FUNCTION BITS_TO_LWORD
  (* Standard: 61499-1 *)
  (* Version 1.0, 2024-02-22, franz *)
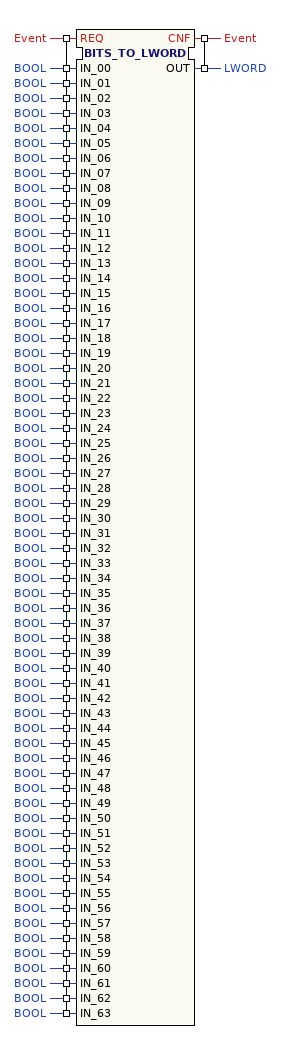
  EVENT_INPUT
    REQ WITH IN_00, IN_01, IN_02, IN_03, IN_04, IN_05, IN_06, IN_07, IN_08, IN_09, IN_10, IN_11, IN_12, IN_13, IN_14, IN_15, IN_16, IN_17, IN_18, IN_19, IN_20, IN_21, IN_22, IN_23, IN_24, IN_25, IN_26, IN_27, IN_28, IN_29, IN_30, IN_31, IN_32, IN_33, IN_34, IN_35, IN_36, IN_37, IN_38, IN_39, IN_40, IN_41, IN_42, IN_43, IN_44, IN_45, IN_46, IN_47, IN_48, IN_49, IN_50, IN_51, IN_52, IN_53, IN_54, IN_55, IN_56, IN_57, IN_58, IN_59, IN_60, IN_61, IN_62, IN_63;
  END_EVENT
  EVENT_OUTPUT
    CNF WITH OUT;
  END_EVENT
  VAR_INPUT
    IN_00 : BOOL; (* BIT 00 *)
    IN_01 : BOOL; (* BIT 01 *)
    IN_02 : BOOL; (* BIT 02 *)
    IN_03 : BOOL; (* BIT 03 *)
    IN_04 : BOOL; (* BIT 04 *)
    IN_05 : BOOL; (* BIT 05 *)
    IN_06 : BOOL; (* BIT 06 *)
    IN_07 : BOOL; (* BIT 07 *)
    IN_08 : BOOL; (* BIT 08 *)
    IN_09 : BOOL; (* BIT 09 *)
    IN_10 : BOOL; (* BIT 10 *)
    IN_11 : BOOL; (* BIT 11 *)
    IN_12 : BOOL; (* BIT 12 *)
    IN_13 : BOOL; (* BIT 13 *)
    IN_14 : BOOL; (* BIT 14 *)
    IN_15 : BOOL; (* BIT 15 *)
    IN_16 : BOOL; (* BIT 16 *)
    IN_17 : BOOL; (* BIT 17 *)
    IN_18 : BOOL; (* BIT 18 *)
    IN_19 : BOOL; (* BIT 19 *)
    IN_20 : BOOL; (* BIT 20 *)
    IN_21 : BOOL; (* BIT 21 *)
    IN_22 : BOOL; (* BIT 22 *)
    IN_23 : BOOL; (* BIT 23 *)
    IN_24 : BOOL; (* BIT 24 *)
    IN_25 : BOOL; (* BIT 25 *)
    IN_26 : BOOL; (* BIT 26 *)
    IN_27 : BOOL; (* BIT 27 *)
    IN_28 : BOOL; (* BIT 28 *)
    IN_29 : BOOL; (* BIT 29 *)
    IN_30 : BOOL; (* BIT 30 *)
    IN_31 : BOOL; (* BIT 31 *)
    IN_32 : BOOL; (* BIT 32 *)
    IN_33 : BOOL; (* BIT 33 *)
    IN_34 : BOOL; (* BIT 34 *)
    IN_35 : BOOL; (* BIT 35 *)
    IN_36 : BOOL; (* BIT 36 *)
    IN_37 : BOOL; (* BIT 37 *)
    IN_38 : BOOL; (* BIT 38 *)
    IN_39 : BOOL; (* BIT 39 *)
    IN_40 : BOOL; (* BIT 40 *)
    IN_41 : BOOL; (* BIT 41 *)
    IN_42 : BOOL; (* BIT 42 *)
    IN_43 : BOOL; (* BIT 43 *)
    IN_44 : BOOL; (* BIT 44 *)
    IN_45 : BOOL; (* BIT 45 *)
    IN_46 : BOOL; (* BIT 46 *)
    IN_47 : BOOL; (* BIT 47 *)
    IN_48 : BOOL; (* BIT 48 *)
    IN_49 : BOOL; (* BIT 49 *)
    IN_50 : BOOL; (* BIT 50 *)
    IN_51 : BOOL; (* BIT 51 *)
    IN_52 : BOOL; (* BIT 52 *)
    IN_53 : BOOL; (* BIT 53 *)
    IN_54 : BOOL; (* BIT 54 *)
    IN_55 : BOOL; (* BIT 55 *)
    IN_56 : BOOL; (* BIT 56 *)
    IN_57 : BOOL; (* BIT 57 *)
    IN_58 : BOOL; (* BIT 58 *)
    IN_59 : BOOL; (* BIT 59 *)
    IN_60 : BOOL; (* BIT 60 *)
    IN_61 : BOOL; (* BIT 61 *)
    IN_62 : BOOL; (* BIT 62 *)
    IN_63 : BOOL; (* BIT 63 *)
  END_VAR
  VAR_OUTPUT
    OUT : LWORD; (* LWORD Output *)
  END_VAR
  BODY IN ST:
FUNCTION BITS_TO_LWORD

VAR_INPUT
	IN_00 : BOOL;    // BIT 00
	IN_01 : BOOL;    // BIT 01
	IN_02 : BOOL;    // BIT 02
	IN_03 : BOOL;    // BIT 03
	IN_04 : BOOL;    // BIT 04
	IN_05 : BOOL;    // BIT 05
	IN_06 : BOOL;    // BIT 06
	IN_07 : BOOL;    // BIT 07
	IN_08 : BOOL;    // BIT 08
	IN_09 : BOOL;    // BIT 09
	IN_10 : BOOL;    // BIT 10
	IN_11 : BOOL;    // BIT 11
	IN_12 : BOOL;    // BIT 12
	IN_13 : BOOL;    // BIT 13
	IN_14 : BOOL;    // BIT 14
	IN_15 : BOOL;    // BIT 15
	IN_16 : BOOL;    // BIT 16
	IN_17 : BOOL;    // BIT 17
	IN_18 : BOOL;    // BIT 18
	IN_19 : BOOL;    // BIT 19
	IN_20 : BOOL;    // BIT 20
	IN_21 : BOOL;    // BIT 21
	IN_22 : BOOL;    // BIT 22
	IN_23 : BOOL;    // BIT 23
	IN_24 : BOOL;    // BIT 24
	IN_25 : BOOL;    // BIT 25
	IN_26 : BOOL;    // BIT 26
	IN_27 : BOOL;    // BIT 27
	IN_28 : BOOL;    // BIT 28
	IN_29 : BOOL;    // BIT 29
	IN_30 : BOOL;    // BIT 30
	IN_31 : BOOL;    // BIT 31
	IN_32 : BOOL;    // BIT 32
	IN_33 : BOOL;    // BIT 33
	IN_34 : BOOL;    // BIT 34
	IN_35 : BOOL;    // BIT 35
	IN_36 : BOOL;    // BIT 36
	IN_37 : BOOL;    // BIT 37
	IN_38 : BOOL;    // BIT 38
	IN_39 : BOOL;    // BIT 39
	IN_40 : BOOL;    // BIT 40
	IN_41 : BOOL;    // BIT 41
	IN_42 : BOOL;    // BIT 42
	IN_43 : BOOL;    // BIT 43
	IN_44 : BOOL;    // BIT 44
	IN_45 : BOOL;    // BIT 45
	IN_46 : BOOL;    // BIT 46
	IN_47 : BOOL;    // BIT 47
	IN_48 : BOOL;    // BIT 48
	IN_49 : BOOL;    // BIT 49
	IN_50 : BOOL;    // BIT 50
	IN_51 : BOOL;    // BIT 51
	IN_52 : BOOL;    // BIT 52
	IN_53 : BOOL;    // BIT 53
	IN_54 : BOOL;    // BIT 54
	IN_55 : BOOL;    // BIT 55
	IN_56 : BOOL;    // BIT 56
	IN_57 : BOOL;    // BIT 57
	IN_58 : BOOL;    // BIT 58
	IN_59 : BOOL;    // BIT 59
	IN_60 : BOOL;    // BIT 60
	IN_61 : BOOL;    // BIT 61
	IN_62 : BOOL;    // BIT 62
	IN_63 : BOOL;    // BIT 63
END_VAR

VAR_OUTPUT
	OUT : LWORD;    // LWORD Output
END_VAR

(* this Function combines the 64 Bits to a lword *)
OUT.0 := IN_00;
OUT.1 := IN_01;
OUT.2 := IN_02;
OUT.3 := IN_03;
OUT.4 := IN_04;
OUT.5 := IN_05;
OUT.6 := IN_06;
OUT.7 := IN_07;
OUT.8 := IN_08;
OUT.9 := IN_09;
OUT.10 := IN_10;
OUT.11 := IN_11;
OUT.12 := IN_12;
OUT.13 := IN_13;
OUT.14 := IN_14;
OUT.15 := IN_15;
OUT.16 := IN_16;
OUT.17 := IN_17;
OUT.18 := IN_18;
OUT.19 := IN_19;
OUT.20 := IN_20;
OUT.21 := IN_21;
OUT.22 := IN_22;
OUT.23 := IN_23;
OUT.24 := IN_24;
OUT.25 := IN_25;
OUT.26 := IN_26;
OUT.27 := IN_27;
OUT.28 := IN_28;
OUT.29 := IN_29;
OUT.30 := IN_30;
OUT.31 := IN_31;
OUT.32 := IN_32;
OUT.33 := IN_33;
OUT.34 := IN_34;
OUT.35 := IN_35;
OUT.36 := IN_36;
OUT.37 := IN_37;
OUT.38 := IN_38;
OUT.39 := IN_39;
OUT.40 := IN_40;
OUT.41 := IN_41;
OUT.42 := IN_42;
OUT.43 := IN_43;
OUT.44 := IN_44;
OUT.45 := IN_45;
OUT.46 := IN_46;
OUT.47 := IN_47;
OUT.48 := IN_48;
OUT.49 := IN_49;
OUT.50 := IN_50;
OUT.51 := IN_51;
OUT.52 := IN_52;
OUT.53 := IN_53;
OUT.54 := IN_54;
OUT.55 := IN_55;
OUT.56 := IN_56;
OUT.57 := IN_57;
OUT.58 := IN_58;
OUT.59 := IN_59;
OUT.60 := IN_60;
OUT.61 := IN_61;
OUT.62 := IN_62;
OUT.63 := IN_63;
END_FUNCTION
  END_BODY
END_FUNCTION
